// TwinCAT 3 PLC project PLC
// ProgramVersion: 3.1.4026.20
// libraries:
//   AUT_Utilities, * (AU-tomation)
//   Tc2_Standard, * (Beckhoff Automation GmbH)
//   Tc2_System, * (Beckhoff Automation GmbH)
//   TcUnit, * (www.tcunit.org)
// project tree:
//   / PlcTask.TcTTO (not stored)
//   POUs/ PRG_TEST.TcPOU, StringBuilder_Test.TcPOU (not stored)
// real-time tasks:
//   TASK PlcTask: cycle T#10ms, priority 20, ADS port 350

// ---- POUs/PRG_TEST.TcPOU
PROGRAM PRG_TEST
VAR
    _StringBuilder_Test : StringBuilder_Test;
END_VAR

TcUnit.RUN();

END_PROGRAM
